(* IEC 61131-3 sources: robocpp/examples, 17 files *)

(* ---- aggregates.st ---- *)
TYPE
    Small : INT(0..10);
    Mode : (Idle, Run, Fault);
    Pair : STRUCT
        Low : Small := 1;
        High : Small := 2;
    END_STRUCT;
END_TYPE

PROGRAM Demo
VAR
    Values : ARRAY [1..3] OF Small := [1, 2, 3];
    Window : Pair := (Low := 4, High := 6);
    State : Mode := Idle;
    Total : INT := 0;
    IsRun : BOOL := FALSE;
END_VAR

Values[2] := Values[1] + Window.High;
Window.Low := Values[2];
State := Run;
IsRun := State = Run;
Total := Values[2] + Window.Low;
END_PROGRAM

(* ---- all_data_types.st ---- *)
TYPE
    AxisMode : (Disabled, Homing, Enabled, Faulted);
    Percent : INT(0..100);
    Counts : ARRAY [0..3] OF DINT;
    AxisStatus : STRUCT
        Mode : AxisMode := Disabled;
        Load : Percent := 0;
        Name : STRING[12] := 'axis';
    END_STRUCT;
END_TYPE

PROGRAM AllDataTypes
VAR
    BoolValue : BOOL := BOOL#TRUE;
    SintValue : SINT := SINT#-8;
    IntValue : INT := INT#123;
    DintValue : DINT := DINT#1000;
    LintValue : LINT := LINT#100000;
    UsintValue : USINT := USINT#200;
    UintValue : UINT := UINT#1000;
    UdintValue : UDINT := UDINT#100000;
    UlintValue : ULINT := ULINT#1000000;
    ByteValue : BYTE := BYTE#16#2A;
    WordValue : WORD := WORD#16#00FF;
    DwordValue : DWORD := DWORD#16#0000FFFF;
    LwordValue : LWORD := LWORD#16#00000000000000FF;
    RealValue : REAL := REAL#3.5;
    LrealValue : LREAL := LREAL#2.25;
    Duration : TIME := T#1d2h3m4s5ms;
    Today : DATE := D#2024-02-29;
    Clock : TIME_OF_DAY := TOD#23:59:59.999;
    Stamp : DATE_AND_TIME := DT#2024-02-29-23:59:59.999;
    Text : STRING[32] := STRING#'robot';
    Wide : WSTRING[32] := WSTRING#"axis";
    Mode : AxisMode := AxisMode#Homing;
    Load : Percent := Percent#75;
    Samples : Counts := [4(0)];
    Snapshot : AxisStatus := (Mode := Enabled, Load := 42, Name := 'joint');
END_VAR

BoolValue := NOT BoolValue;
IntValue := SintValue + 10;
DintValue := DintValue + 1;
Samples[1] := DintValue;
Mode := Enabled;
Snapshot.Load := Load;
Text := CONCAT(Text, ' arm');
Wide := WSTRING#"wide";
END_PROGRAM

(* ---- configuration.st ---- *)
PROGRAM ConfiguredProgram
VAR
    Count : INT := 0;
END_VAR

Count := Count + 1;
END_PROGRAM

CONFIGURATION Plant
VAR_GLOBAL
    PlantOffset : INT := 1;
END_VAR
RESOURCE Cpu ON PLC
    VAR_CONFIG
        Tunable AT %MW10 : INT := 5;
    END_VAR
    VAR_ACCESS
        StartAccess AT %MX0.0 : BOOL;
    END_VAR
    TASK Fast(INTERVAL := T#10ms, PRIORITY := 1);
    PROGRAM Main WITH Fast : ConfiguredProgram;
END_RESOURCE
END_CONFIGURATION

(* ---- control_flow.st ---- *)
PROGRAM ControlFlowDemo
VAR
    I : INT := 0;
    Total : INT := 0;
    Selected : INT := 0;
    Done : BOOL := FALSE;
END_VAR

FOR I := 1 TO 3 DO
    Total := Total + I;
END_FOR;

WHILE Total < 8 DO
    Total := Total + 1;
END_WHILE;

REPEAT
    Total := Total - 1;
UNTIL Total = 7
END_REPEAT;

Selected := MAX(Total, 3);

CASE Selected OF
    7: Done := TRUE;
    ELSE Done := FALSE;
END_CASE;
END_PROGRAM

(* ---- conversions.st ---- *)
PROGRAM Demo
VAR
    Text : STRING[32] := '';
    Parsed : INT := 0;
    Truncated : INT := 0;
    Bcd : WORD := 0;
    FromBcd : INT := 0;
    RealValue : REAL := 0.0;
    Flag : BOOL := FALSE;
    Delay : TIME := T#0ms;
END_VAR

Parsed := STRING_TO_INT('42');
Truncated := TRUNC(-1.6);
Bcd := INT_TO_BCD(369);
FromBcd := BCD_TO_INT(Bcd) + WORD_BCD_TO_UINT(UINT_TO_BCD_WORD(25));
RealValue := STRING_TO_REAL('2.5');
Flag := STRING_TO_BOOL('TRUE');
Delay := STRING_TO_TIME('T#250ms') + INT_TO_TIME(50);
Text := CONCAT(BOOL_TO_STRING(Flag), INT_TO_STRING(Parsed));
END_PROGRAM

(* ---- counter.st ---- *)
PROGRAM CounterDemo
VAR
    Count : INT := 0;
    Limit : INT := 3;
    Done : BOOL := FALSE;
END_VAR

IF Count < Limit THEN
    Count := Count + 1;
ELSE
    Done := TRUE;
END_IF;
END_PROGRAM

(* ---- function_blocks.st ---- *)
PROGRAM FunctionBlockDemo
VAR
    Counter : CTU;
    Latch : SR;
    Edge : R_TRIG;
    Pulse : BOOL := FALSE;
    Count : INT := 0;
    CountDone : BOOL := FALSE;
    Latched : BOOL := FALSE;
    Rising : BOOL := FALSE;
END_VAR

Pulse := NOT Pulse;
Counter(CU := Pulse, R := FALSE, PV := 2);
Latch(S1 := Counter.Q, R := FALSE);
Edge(CLK := Pulse);

Count := Counter.CV;
CountDone := Counter.Q;
Latched := Latch.Q1;
Rising := Edge.Q;
END_PROGRAM

(* ---- functions.st ---- *)
FUNCTION Scale : INT
VAR_INPUT
    Input : INT;
    Factor : INT;
END_VAR

Scale := Input * Factor;
END_FUNCTION

PROGRAM FunctionDemo
VAR
    A : INT := 4;
    B : INT := 0;
    C : INT := 0;
END_VAR

B := Scale(A, 3);
C := Scale(Input := B, Factor := 2);
END_PROGRAM

(* ---- instruction_list.il ---- *)
PROGRAM InstructionListFile
VAR
    A : INT := 3;
    B : INT := 4;
    Sum : INT := 0;
    Bigger : BOOL := FALSE;
END_VAR

LD A
ADD B
ST Sum
LD Sum
GT 5
ST Bigger
END_PROGRAM

(* ---- instruction_list.st ---- *)
PROGRAM InstructionListDemo
VAR
    A : INT := 3;
    B : INT := 4;
    C : INT := 0;
    Bigger : BOOL := FALSE;
    Complex : BOOL := FALSE;
END_VAR

LD A;
ADD B;
ST C;
GT 5;
ST Bigger;
LD TRUE;
AND (Bigger OR FALSE);
ST Complex;
END_PROGRAM

(* ---- instruction_list_calls.st ---- *)
PROGRAM Demo
VAR
    Counter : CTU;
    Done : BOOL := FALSE;
    Cv : INT := 0;
    Skipped : INT := 0;
END_VAR

LD TRUE;
CALC Counter(CU := TRUE, R := FALSE, PV := 1);
LD Counter.Q;
ST Done;
LD Counter.CV;
ST Cv;
LD TRUE;
RETC;
Skipped := 1;
END_PROGRAM

(* ---- instruction_list_jumps.st ---- *)
PROGRAM IlJumpDemo
VAR
    Count : INT := 0;
    Done : BOOL := FALSE;
END_VAR

LD Count;
GE 3;
JMPC DoneLabel;
LD Count;
ADD 1;
ST Count;
JMP EndLabel;

DoneLabel:
LD TRUE;
ST Done;

EndLabel:
END_PROGRAM

(* ---- sfc_qualifiers.st ---- *)
PROGRAM Qualifiers
VAR
    PulseCount : INT := 0;
    DelayCount : INT := 0;
    LimitCount : INT := 0;
END_VAR

INITIAL_STEP Pulse;
STEP Delay;
STEP Limit;
TRANSITION ToDelay := PulseCount >= 1;
TRANSITION ToLimit := DelayCount >= 1;
ACTION Pulse(P):
    PulseCount := PulseCount + 1;
END_ACTION;
ACTION Delay(D, T#2ms):
    DelayCount := DelayCount + 1;
END_ACTION;
ACTION Limit(L, T#2ms):
    LimitCount := LimitCount + 1;
END_ACTION;
END_PROGRAM

(* ---- sfc_sequence.st ---- *)
PROGRAM Sequence
VAR
    Ready : BOOL := TRUE;
    Done : BOOL := FALSE;
END_VAR

INITIAL_STEP Start;
STEP Run;
TRANSITION Go := Ready;
ACTION Run:
    Done := TRUE;
END_ACTION;
END_PROGRAM

(* ---- st_bit_ops.st ---- *)
PROGRAM Demo
VAR
    Mask : INT := 0;
    Inverted : INT := 0;
    Flag : BOOL := FALSE;
END_VAR

Mask := (15 AND 51) OR (1 XOR 3);
Inverted := NOT 15;
Flag := (TRUE AND FALSE) OR TRUE;
END_PROGRAM

(* ---- strings_dates.st ---- *)
PROGRAM Demo
VAR
    Text : STRING[16] := 'robot';
    Out : STRING[16] := '';
    Found : INT := 0;
    Today : DATE := D#1970-01-02;
    Noon : TIME_OF_DAY := TOD#12:00:00.250;
    Stamp : DATE_AND_TIME := DT#1970-01-02-00:00:01;
END_VAR

Out := CONCAT(LEFT(Text, 2), RIGHT('code', 2));
Found := FIND(INSERT('ro', 'bo', 2), 'bo');
END_PROGRAM

(* ---- timers.st ---- *)
PROGRAM TimerDemo
VAR
    Delay : TON;
    Pulse : TP;
    Done : BOOL := FALSE;
    PulseActive : BOOL := FALSE;
    Elapsed : TIME := T#0ms;
END_VAR

Delay(IN := TRUE, PT := T#2ms);
Pulse(IN := TRUE, PT := T#2ms);

Done := Delay.Q;
PulseActive := Pulse.Q;
Elapsed := Delay.ET;
END_PROGRAM
